// TIA Portal V19 export
VAR_GLOBAL   // PLC tag table "TT - Loading"
   iLoadingSenDown_a1 AT %I0.4 : Bool;
   iLoadingSenUp_a0 AT %I0.5 : Bool;
   iLoadingSenAtPick_b0 AT %I0.6 : Bool;
   iLoadingSenAtPlace_b1 AT %I0.7 : Bool;
   "oLoadingVenCilDown_A+" AT %Q0.1 : Bool;
   oLoadingVenCilPlace_B AT %Q0.2 : Bool;
   oLoadingVenGrip_C AT %Q0.3 : Bool;
END_VAR
